{attribute 'qualified_only'}
VAR_GLOBAL
	bButtonWinderPower			: BOOL := TRUE;
	bButtonStartWinder			: BOOL;
	bButtonStopWinder			: BOOL;
	bButtonResetWinder			: BOOL;
	bButtonWinderDirection		: BOOL;
	bButtonNotWinderDirection	: BOOL;
	bButtonSelectionMode		: BOOL;
	bButtonSetupMode			: BOOL;
	bButtonManualMode			: BOOL;
	bButtonProdutionMode 		: BOOL;
	ActTapeSpeed				: REAL;
	ActTorque					: LREAL;
	RunningLength				: REAL;
END_VAR

(* stored: Version 1.1.0.1
   GVL GVL_HMI: Id {55c4c117-0c12-4f72-9e54-90272aed3981} *)
